Staubli VAL3: Day2.dtx

mdesc mNomSpeed
string sInput
num nInput
lists lResult
  [0]
    string sString
string sCommand
num nValue
string sValue
